INTERFACE IScribly EXTENDS ZApplication.IUnit

END_INTERFACE

(* stored: Version 1.1.0.1
   Itf IScribly: Id {0b4fb60c-e5d9-47a6-85d8-a573a03570d0} *)
